FUNCTION F_SendEvent : BOOL

VAR_INPUT
	Event			: StatsEvent;
END_VAR

VAR_IN_OUT
	StatsFIFO		: FIFO_StatsEvent;
	Buffer			: StatsEventFIFOBuffer;
END_VAR

VAR
	TempEvent		: StatsEvent;
END_VAR

VAR_EXTERNAL
	gCurrentTime	: TimeStamp;	// Global System Time Variable
END_VAR

// Use Temp Event, Update TimeStamp
TempEvent := Event;
TempEvent.TimeStamp := gCurrentTime;

// Load Event to Stats FIFO
StatsFIFO(pFIFO := ADR(Buffer));
StatsFIFO.LOAD(Input := TempEvent);

END_FUNCTION

(* stored: Version 1.1.0.1, ProductVersion 3.1.4024.9
   POU F_SendEvent: Id {12d18f17-aa0f-416e-b681-8ce260ed3d31}, SpecialFunc None *)
